// TIA Portal V17 export
// export: Created 2026-04-13T11:12:42.4476824Z, ExportSetting WithDefaults, DisplayName Totally Integrated Automation Portal, DisplayVersion V17 Update 4, DisplayName TIA Portal Openness, DisplayVersion V17 Update 4, DisplayName TIA Portal Version Control Interface, DisplayVersion V17, DisplayName SINAMICS Startdrive Advanced, DisplayVersion V17, DisplayName SINAMICS Startdrive G130, G150, S120, S150, SINAMICS MV, S210, DisplayVersion V17, DisplayName SINAMICS Startdrive G110M, G120, G120C, G120D, G120P, G115D, DisplayVersion V17, DisplayName STEP 7 Professional, DisplayVersion V17 Update 4, DisplayName STEP 7 Safety, DisplayVersion V17, DisplayName WinCC Professional, DisplayVersion V17 Update 4
FUNCTION_BLOCK "3-延时开关S"   // FB73, SCL
{ S7_Optimized_Access := 'TRUE' }
VERSION : 0.1
// stored: AutoNumber true, IsIECCheckEnabled false, IsRetainMemResEnabled false, MemoryReserve 100, SetENOAutomatically false, UDAEnableTagReadback false
   VAR_INPUT
      B_IN : Bool;   // 启动/关闭信号输入
      T_IN : Int;   // 延时时间(单位:秒)
      B_Status : Bool;   // 运行状态
   END_VAR
   VAR_OUTPUT
      B_OUT : Bool;   // 启动/关闭信号输出
   END_VAR
   VAR
      R_TRIG_1 { S7_SetPoint := 'True'} : R_TRIG;   // 计时_1S
      i : UDInt;
   END_VAR
BEGIN
   (*水泵关机延时功能:
       1.立即开机
       2.延时I_IN分钟后关闭
       3.延时关机期间如果水泵手动/其他原因关闭,延时时间清零,立即关闭
   *)

   #R_TRIG_1(CLK:="Clock_1Hz");

   IF NOT #B_IN THEN
       IF #R_TRIG_1.Q THEN
           #i += 1;
       END_IF;
   ELSE
       #i := 0;
   END_IF;

   IF #B_IN THEN
       #B_OUT := 1;    //立即开
   ELSIF NOT #B_IN AND #i >= #T_IN  THEN    //延时关
       #B_OUT := 0;
   ELSIF NOT #B_IN AND #i < #T_IN  AND  #B_Status THEN  //延时关机期间如果水泵手动/其他原因关闭,延时时间清零,立即关闭
       #B_OUT := 0;
   END_IF;
END_FUNCTION_BLOCK
